FUNCTION_BLOCK FB_BlueFlag
VAR_INPUT
	Bnt_Blueflag: BOOL;	// 接带输入信号
	FlagDone: BOOL;// 电芯下料完成信号
	AixsoActPos: LREAL;//放卷轴当前角度
	Diameter: REAL;//放卷轴当前卷径
	SetLenght: REAL;//接带点到叠台的距离
	fYDLength: LREAL;
	rBnt_BlueflagCaNum: UINT;
END_VAR
VAR_OUTPUT
		FlagPoisn: ARRAY[0..20]OF BOOL;
END_VAR
VAR
	rBnt_Blueflag: R_TRIG;
	rFlagDone: R_TRIG;
	i: INT;
	RemberPos: ARRAY[0..20] OF LREAL;
	RemberPos1: ARRAY[0..20] OF LREAL;
	RemberPos2: ARRAY[0..20] OF LREAL;
END_VAR

VAR_IN_OUT
	rBnt_BlueflagNum: UINT;
	rBnt_Blueflaging: BOOL;	
	NumberPos: ARRAY[0..20] OF LREAL;//接带点记录数据
	NumberPos1: ARRAY[0..20] OF LREAL;//接带点记录数据
	NumberPos2: ARRAY[0..20] OF LREAL;//接带点记录数据
END_VAR

rBnt_Blueflag(CLK:=Bnt_Blueflag , Q=> );	// 接带输入信号
rFlagDone(CLK:=FlagDone , Q=> );	// 电芯下料完成信号
//根据接带信号记录放卷轴当前的角度
IF rBnt_Blueflag.Q THEN
		rBnt_Blueflaging:=TRUE;//接带信号
		rBnt_BlueflagNum:=rBnt_BlueflagCaNum;
		FOR i:=0 TO 20 BY 1 DO
							IF i<20 THEN
									NumberPos[20-i]:=	NumberPos[19-i];
							ELSE
									NumberPos[0]:=AixsoActPos;
							END_IF;
							
							IF i<20 THEN
									NumberPos1[20-i]:=	NumberPos1[19-i];
							ELSE
									NumberPos1[0]:=AixsoActPos+fYDLength;
							END_IF;
							
							IF i<20 THEN
									NumberPos2[20-i]:=	NumberPos2[19-i];
							ELSE
									NumberPos2[0]:=AixsoActPos+fYDLength*2;
							END_IF;
		END_FOR
END_IF
//根据当前的角度
FOR i:=0 TO 20 BY 1 DO
		IF NumberPos[i]<>0 THEN
			RemberPos[i]:= FC_AngleToLength(ABS(AixsoActPos-NumberPos[i]),Diameter);			
		END_IF
		
		IF NumberPos1[i]<>0 THEN
			RemberPos1[i]:= FC_AngleToLength(ABS(AixsoActPos-NumberPos1[i]),Diameter);
		END_IF
		
		IF NumberPos2[i]<>0 THEN
			RemberPos2[i]:= FC_AngleToLength(ABS(AixsoActPos-NumberPos2[i]),Diameter);
		END_IF

		IF (RemberPos[i] >= SetLenght AND NumberPos[i]<>0) OR (RemberPos1[i] >= SetLenght AND NumberPos1[i]<>0)OR (RemberPos2[i] >= SetLenght AND NumberPos2[i]<>0)   THEN
			FlagPoisn[i]:=TRUE;
		END_IF
		
		IF (RemberPos[i] >= SetLenght AND NumberPos[i]<>0) AND rFlagDone.Q THEN
			FlagPoisn[i] :=FALSE;
			NumberPos[i]:=0;
		END_IF
	
		IF (RemberPos1[i] >= SetLenght AND NumberPos1[i]<>0) AND rFlagDone.Q THEN
			FlagPoisn[i] :=FALSE;
			NumberPos1[i]:=0;
		END_IF	

		IF (RemberPos2[i] >= SetLenght AND NumberPos2[i]<>0) AND rFlagDone.Q THEN
			FlagPoisn[i] :=FALSE;
			NumberPos2[i]:=0;
		END_IF		
END_FOR

END_FUNCTION_BLOCK

(* stored: Version 1.1.0.1, ProductVersion 3.1.4024.9
   POU FB_BlueFlag: Id {f6ad9ecd-ec40-48a0-ada6-07b4ae66e860}, SpecialFunc None *)
